# EPICS substitutions: epics/ioc/PinholeMotionTop/iocBoot/iocHorizontalZaber/horizontal.zaber.substitutions
file "$(MOTOR)/motorApp/Db/asyn_motor.db"
{
  pattern
  {P,                            N,   M,         DTYP,                      PORT,   ADDR,           DESC,                     EGU,   DIR,   VELO,  VBAS, ACCL,  BDST, BVEL, BACC,   MRES, PREC,    DLLM,   DHLM, INIT}
  {Beamline:DivergencePinhole:,  1,   H,  "asynMotor",     DivergencePinholeHPort,     0,   "Divergence pinhole horizontal",   mm,   Pos,  100.0,   5.0,   .5,     0,    1,   .2,  0.001,    3,       0,    150,   ""}
  {Beamline:EnergyPinhole:,      1,   H,  "asynMotor",     EnergyPinholeHPort,         0,   "Energy pinhole horizontal",       mm,   Pos,  100.0,   5.0,   .5,     0,    1,   .2,  0.001,    3,       0,    150,   ""}
}
